SUBAPPLICATION Button_Aux_IE (* Button (nicht-latching) ODER AUX-Zuweisung (Joystick) aktiviert -> 1 gemeinsames IND-Event (BT_RELEASED_UNLATCHED bzw. AuxEnabled fest verdrahtet). Analog Softkey_Aux_IE, aber fuer einen echten VT-Button (Klasse CButton) statt eines SoftKeys - Softkey_IE und Button_IE sind zwei getrennte FORTE-Service-Interface-Bausteine fuer unterschiedliche VT-Activation-Messages, ein Button liefert NIE ein SK_PRESSED (Franz, 2026-09-20, hat Softkey_IE selbst implementiert: 'tut sie NICHT'). Der Button MUSS non-latching sein (Latchable=0 im Pool) - ein latching Button kann nur sinnvoll ueber Button_IXA (Dauerzustand/Pegel) gelesen werden, nicht ueber dieses Event-InputEvent-Muster (Franz, 2026-09-20). *)
  (* Standard: 61499-2; Description: Copyright (c) 2026 Meisterschulen am Ostbahnhof This program and the accompanying materials are made available under the terms of the Eclipse Public License 2.0 which is available at https://www.eclipse.org/legal/epl-2.0/ SPDX-License-Identifier: EPL-2.0 *)
  (* Version 1.0, 2026-09-20, Franz Höpfinger, Meisterschulen am Ostbahnhof, initial implementation - Bugfix fuer Automatik_Toggle_Button.SUB (nutzte bisher Softkey_Aux_IE mit einer Button-Object-ID, Softkey_IE empfaengt aber keine Button-Activation-Message - bestaetigt vom Autor der FORTE-Implementierung). *)
  PACKAGE MyLib::sys;
  IMPORT isobus::UT::io::Button::ButtonActivationCode::BT_RELEASED_UNLATCHED;
  IMPORT isobus::UT::io::Auxiliary::IN::AuxiliaryState::AuxDisabled_START;
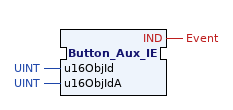
  EVENT_OUTPUT
    IND; (* Feuert wenn Button (BT_RELEASED_UNLATCHED) ODER Aux (AuxEnabled) aktiviert wird *)
  END_EVENT
  VAR_INPUT
    u16ObjId : UINT; (* Object ID Button (CButton, non-latching) *)
    u16ObjIdA : UINT; (* Object ID AuxFunction2 *)
  END_VAR
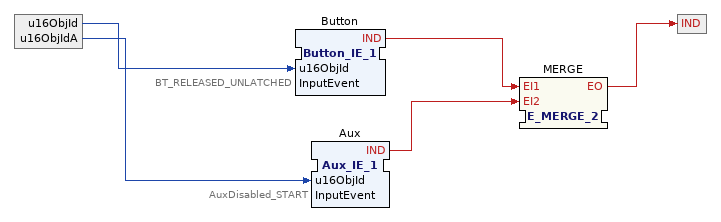
  FBS
    MERGE : iec61499::events::E_MERGE_2;
  END_FBS
  SUBAPPS
    Button : MyLib::sys::Button_IE_1(InputEvent := BT_RELEASED_UNLATCHED);
    Aux : MyLib::sys::Aux_IE_1(InputEvent := AuxDisabled_START);
  END_SUBAPPS
  EVENT_CONNECTIONS
    Button.IND TO MERGE.EI1;
    Aux.IND TO MERGE.EI2;
    MERGE.EO TO IND;
  END_CONNECTIONS
  DATA_CONNECTIONS
    u16ObjId TO Button.u16ObjId;
    u16ObjIdA TO Aux.u16ObjId;
  END_CONNECTIONS
END_SUBAPPLICATION
